# B&R Automation Studio project ABC_Pltzr (part 2)

#### Cyclic.ld
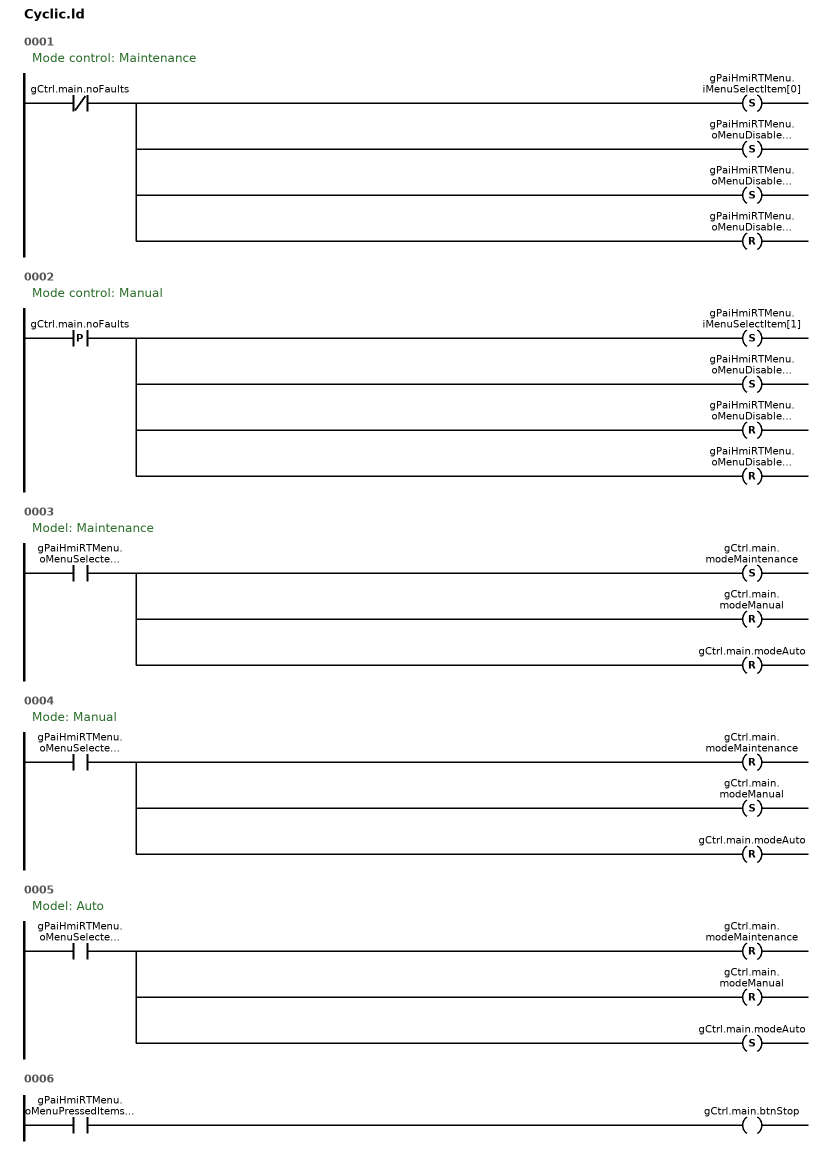
Ladder, written as Structured Text:
```iecst
PROGRAM _CYCLIC
VAR
    _e1 : R_TRIG;
END_VAR
(* Network 1: Mode control: Maintenance *)
IF NOT gCtrl.main.noFaults THEN
    gPaiHmiRTMenu.iMenuSelectItem[0] := TRUE;
    gPaiHmiRTMenu.oMenuDisabledItems[1] := TRUE;
    gPaiHmiRTMenu.oMenuDisabledItems[2] := TRUE;
    gPaiHmiRTMenu.oMenuDisabledItems[0] := FALSE;
END_IF;

(* Network 2: Mode control: Manual *)
_e1(CLK := gCtrl.main.noFaults);
IF _e1.Q THEN
    gPaiHmiRTMenu.iMenuSelectItem[1] := TRUE;
    gPaiHmiRTMenu.oMenuDisabledItems[0] := TRUE;
    gPaiHmiRTMenu.oMenuDisabledItems[1] := FALSE;
    gPaiHmiRTMenu.oMenuDisabledItems[2] := FALSE;
END_IF;

(* Network 3: Model: Maintenance *)
IF gPaiHmiRTMenu.oMenuSelectedItems[0] THEN
    gCtrl.main.modeMaintenance := TRUE;
    gCtrl.main.modeManual := FALSE;
    gCtrl.main.modeAuto := FALSE;
END_IF;

(* Network 4: Mode: Manual *)
IF gPaiHmiRTMenu.oMenuSelectedItems[1] THEN
    gCtrl.main.modeMaintenance := FALSE;
    gCtrl.main.modeManual := TRUE;
    gCtrl.main.modeAuto := FALSE;
END_IF;

(* Network 5: Model: Auto *)
IF gPaiHmiRTMenu.oMenuSelectedItems[2] THEN
    gCtrl.main.modeMaintenance := FALSE;
    gCtrl.main.modeManual := FALSE;
    gCtrl.main.modeAuto := TRUE;
END_IF;

(* Network 6 *)
gCtrl.main.btnStop := gPaiHmiRTMenu.oMenuPressedItems[1];
END_PROGRAM
```

- Program Logical/MachineControl/palletinfauto (IEC) (no source held here)

### Program Logical/paiComponents/bglib

#### bgBitUtilities.h
```c
/**\file: bgBitUtilities.h
*Bit utilities.
*/
#include <bur/plctypes.h>
#ifndef _BG_BITUTILS_H
#define _BG_BITUTILS_H

/**
Set UDINT bits.
\param dest,  Ptr to UDINT.
\param bitIndex within the above UDINT
\param bitValue is the value to set the bit to
*/
void bgBitSetUDINT(UDINT* dest,  UINT bitIndex, BOOL bitValue);

/**
Set UINT bits.
\param dest,  Ptr to UINT.
\param bitIndex within the above UINT
\param bitValue is the value to set the bit to
*/
void bgBitSetUINT(UINT* dest,  UINT bitIndex, BOOL bitValue);

/**
Set USINT bits.
\param dest,  Ptr to USINT.
\param bitIndex within the above USINT
\param bitValue is the value to set the bit to
*/
void bgBitSetUSINT(USINT* dest,  UINT bitIndex, BOOL bitValue);

#endif
```

#### bgPVSerialize.h
```c
/**\file: bgPVSerialize.h
*Serialize/deserialize a PV to/from text stream.
*/
#include <bur/plctypes.h>
#ifndef _BG_PVSERIALIZE_H
#define _BG_PVSERIALIZE_H

/**
Serialize a PV (*pvNameRoot) to an output stream (* toOutStream) with a max length of (lengthOutStream).
\param pvNameRoot ptr to a PV name
\param toOutStream ptr to an output stream (i.e. char buffer)
\param lengthOutStream max length of the output stream in bytes
\return -1 error
\return >=0 number of bytes written to the output stream
*/
DINT bgPVStructSerialize(char* pvNameRoot, char* toOutStream, UDINT lengthOutStream);

/**
Deserialize a PV (*pvNameRoot) from an input stream (* fromStream) that contains (lengthStream) of valid text data.
\param pvNameRoot ptr to a PV name
\param fromStream ptr to an input stream (i.e. char buffer)
\param lengthStream length of the content in the input stream in bytes
\return -1 error
\return >=0 TODO
*/
DINT bgPVStructDeserialize(char* pvNameRoot, char* fromStream, UDINT lengthStream);

/**
Compare two instances of the same structure type using PV services and provide diff report into the given output stream (* toOutStream) with a max length of (lengthOutStream).
\param pvNameRoot ptr to an instance 1 of the PV structure
\param pvNameRoot2 ptr to an instance 2 of the PV structure
\param toOutStream ptr to an output stream (i.e. char buffer)
\param lengthOutStream max length of the output stream in bytes
\return -1 error
\return >=0 number of bytes written to the output stream
*/
DINT bgPVStructCompare(char* pvNameRoot, char* pvNameRoot2, char* toOutStream, UDINT lengthOutStream);

#endif
```

#### bgHttpAppXmlRpc.c
```c
/**\file bgHttpAppXmlRpc.c
*/

#ifndef WIN32
/*
B&R components:
===============================================================================
*/
#include <bur/plc.h>
#include <bur/plctypes.h>
#include <astcp.h>
#include <brsystem.h>
#include <sys_lib.h>
#endif

/*
BG components
===============================================================================
*/
#include "bgdebug.h"
#include "bgstring.h"
#include "bgsscanf.h"
#include "bgTcpSocketClientServer.h"
#include "bgHttpProtocol.h"
#include "bgHttpAppXmlRpc.h"
#include "bgDataStructures.h"
#include "bgBufMemAlloc.h"
#include "bgXmlRpcParser.h"

static void apndXmlBlockOpen(bgTcpSocketSession_typ* pSession, char* keywName);
static void apndXmlBlockClos(bgTcpSocketSession_typ* pSession, char* keywName);

/*
XmlRpc Server
######################################################################################################
######################################################################################################
######################################################################################################
######################################################################################################
*/
void bgXmlRpcServerApplication(bgTcpSocketSession_typ* pSession)
{
char* pMem;
int sizeMem;
char* pMemTree;
int sizeMemTree;
char* pMemStr;
int sizeMemStr;

httpAppXmlRpc_typ* pXmlRpcAppData;
bgXmlRpcParser_typ* pXmlRpc;
bgTree4C_typ* pTree;
bgTree4CNode_typ* pNode;
bgStringHeap_typ* pStrHeap;

int i;

	if( bgXmlRpcServerAppCommon(pSession) ){
		/*common XMLRPC check(s) have failed > exit (& send automatic error response)*/
		return;
	}

/*App Specific Buf MemAlloc*/
	/*1) application specific data structure*/
	if( bgBufMemAllocCreateBlock(&pSession->sessionMem, sizeof(httpAppXmlRpc_typ) + sizeof(char*), &pMem, &sizeMem) )
	{
    	DBGMSG("bgXmlRpcServerApplication(): FATAL ERROR (1); No memory\r\n");
		return;
	}

	pXmlRpcAppData = (httpAppXmlRpc_typ*)pMem;
	pXmlRpc = &pXmlRpcAppData->xmlRpcData;
	pTree = &pXmlRpc->xmlTree;
	pStrHeap = &pXmlRpc->strHeap;

	/*2) set storage for xmlrpc node tree*/
	if( bgBufMemAllocCreateBlock(&pSession->sessionMem, 1500, &pMemTree, &sizeMemTree) )
	{
    	DBGMSG("bgXmlRpcServerApplication(): FATAL ERROR (2); No memory\r\n");
		return;
	}

	/*3) set storage for xmlrpc string heap (rest of the available mem)*/
	if( bgBufMemAllocCreateBlock(&pSession->sessionMem, 0, &pMemStr, &sizeMemStr) )
	{
    	DBGMSG("bgXmlRpcServerApplication(): FATAL ERROR (3); No memory\r\n");
		return;
	}

	DBGMSG("bgXmlRpcServerApplication: memTotal=%d, memData=%d, memTree=%d, memStr=%d\n",
		sizeMem + sizeMemStr + sizeMemTree, sizeMem, sizeMemTree, sizeMemStr);

    bgXmlRpcParserInit(pXmlRpc, bgHttpGetContentStartAddr(pSession), pMemTree, sizeMemTree, pMemStr, sizeMemStr);

    bgXmlRpcParserParse(pXmlRpc);

	if(pXmlRpc->error){
		DBGMSG("xml parsing error=%d; keyword=[%s], line=%d, col=%d)\n",
			pXmlRpc->error,
			bgXmlRpcGetKeywordStr(pXmlRpc->keywId),
			pXmlRpc->keywLineNo,
			pXmlRpc->keywColNo);
/*
			bgXmlRpcServerSendFaultResponse(pSession, 100, "This is fault!");
			rerurn;
*/
	}

    DBGMSG("xmlRpc tree:\n");
    DBGMSG("---------------------------------------------------------------------\n");

    bgTree4CPrint(pTree);

    DBGMSG("---------------------------------------------------------------------\n");

    DBGMSG("xmlRpc list of values:\n");
    DBGMSG("---------------------------------------------------------------------\n");

	for(i=0; i < pTree->nodeCountUsed; i++){

		pNode = &pTree->nodes[i];

		if(!pNode || !pNode->used)
			continue;

		switch(pNode->dataType){
			case XMLRPC_ID_METHOD_NAME:
				DBGMSG("MethodName:[%s]\n", pNode->data ? pNode->data : "unknown");
			break;
			case XMLRPC_ID_NAME:
				DBGMSG("\nParamName:[%s]\n", pNode->data ? pNode->data : "unknown");
			break;
			case XMLRPC_ID_I4:
			case XMLRPC_ID_INT:
			case XMLRPC_ID_BOOL:
				DBGMSG("Value:[%d]\n", pNode->dataValue );

			break;
			case XMLRPC_ID_STRING:
			case XMLRPC_ID_TIME:
				DBGMSG("Value:[%s]\n", pNode->data ? pNode->data : "unknown" );
			break;
			case XMLRPC_ID_DOUBLE:
				DBGMSG("Value:[%f]\n", (float)pNode->dataValue);
			break;
			default:
			break;
		}

	}
    DBGMSG("---------------------------------------------------------------------\n");

	DBGMSG("StringHeap space: total=%d, free=%d\n", pStrHeap->memSize, pStrHeap->memFree );

	bgXmlRpcServerSendFaultResponse(pSession, 100, "This is fault!");
}

int bgXmlRpcServerAppCommon(bgTcpSocketSession_typ* pSession)
{
    /*session/application/protocol specific data structure*/
    httpMessage_typ* r = (httpMessage_typ*)pSession->pProtocol;

	if( r->commandId != BGHTTP_REQUEST_COMMAND_POST){
		DBGMSG("bgXmlRpcServerApplication(): command (%s) not supported!\r\n", r->command);
		bgHttpSendErrorResponse(pSession, 405);
 		return 1;
	}

	return 0;
}

int bgXmlRpcServerSendFaultResponse(bgTcpSocketSession_typ* p, int faultCode, char* faultString)
{
/*
XML-RPC Fault Response Example:

HTTP/1.1 200 OK
Connection: close
Content-Length: 426
Content-Type: text/xml
Date: Fri, 17 Jul 1998 19:55:02 GMT
Server: UserLand Frontier/5.1.2-WinNT

<?xml version="1.0"?>
<methodResponse>
	<fault>
		<value>
			<struct>
				<member>
					<name>faultCode</name>
					<value><int>4</int></value>
				</member>
				<member>
					<name>faultString</name>
					<value><string>Too many parameters.</string></value>
				</member>
			</struct>
		</value>
	</fault>
</methodResponse>
*/
	bgHttpServerSendResponseBeg(p, 200, "text/xml");

	apndXmlBlockOpen(p, XMLRPC_STR_XMLHEADLINE );

	apndXmlBlockOpen(p, XMLRPC_STR_METHOD_RSP);
		apndXmlBlockOpen(p, XMLRPC_STR_FAULT);
			apndXmlBlockOpen(p, XMLRPC_STR_VALUE);
				apndXmlBlockOpen(p, XMLRPC_STR_STRUCT);
					apndXmlBlockOpen(p, XMLRPC_STR_MEMBER);
					{
						char txtBuffer[255];
						bgsprintf(&txtBuffer[0], "<%s>%s</%s>", XMLRPC_STR_NAME, "faultCode", XMLRPC_STR_NAME);
						bgHttpSendBufApndContentLine(p, &txtBuffer[0]);

						bgsprintf(&txtBuffer[0], "<%s><%s>%d</%s></%s>", XMLRPC_STR_VALUE, XMLRPC_STR_INT, faultCode, XMLRPC_STR_INT, XMLRPC_STR_VALUE);
						bgHttpSendBufApndContentLine(p, &txtBuffer[0]);

					}
					apndXmlBlockClos(p, XMLRPC_STR_MEMBER);
					apndXmlBlockOpen(p, XMLRPC_STR_MEMBER);
					{
						char txtBuffer[255];
						bgsprintf(&txtBuffer[0], "<%s>%s</%s>", XMLRPC_STR_NAME, "faultString", XMLRPC_STR_NAME);
						bgHttpSendBufApndContentLine(p, &txtBuffer[0]);

						bgsprintf(&txtBuffer[0], "<%s><%s>%s</%s></%s>", XMLRPC_STR_VALUE, XMLRPC_STR_STRING, faultString, XMLRPC_STR_STRING, XMLRPC_STR_VALUE);
						bgHttpSendBufApndContentLine(p, &txtBuffer[0]);

					}
					apndXmlBlockClos(p, XMLRPC_STR_MEMBER);
				apndXmlBlockClos(p, XMLRPC_STR_STRUCT);
			apndXmlBlockClos(p, XMLRPC_STR_VALUE);
		apndXmlBlockClos(p, XMLRPC_STR_FAULT);
	apndXmlBlockClos(p, XMLRPC_STR_METHOD_RSP );

	bgHttpServerSendResponseEnd(p);
	return 0;
}

int bgXmlRpcServerSendResponse(bgTcpSocketSession_typ* pSession, char* pContent, int contentSize)
{
    bgHttpServerSendResponse(pSession, 200, pContent, contentSize, "text/xml");
	return 0;
}

/*
XmlRpc Client
######################################################################################################
######################################################################################################
######################################################################################################
######################################################################################################
*/
void bgXmlRpcClientSetConnection(bgTcpSocketClient_typ* pClient, char* serverIpAddr, int serverPortNumber)
{
	bgHttpClientSetConnection(pClient, serverIpAddr, serverPortNumber);
}

void bgXmlRpcClientSendRequest(bgTcpSocketClient_typ* pClient, char* pContent , int contentSize)
{
	bgHttpClientSendRequest(pClient, "POST /RPC2 ", pContent , contentSize, "text/xml");
}

void bgXmlRpcClientApplication(bgTcpSocketSession_typ* pSession)
{
int i;
char* pMem;
int sizeMem;
httpAppWeb_typ* pWebData;
int sizeMemAppTotal = 0;

/*App Specific Buf MemAlloc*/
	/*1) application specific data structure*/
	if( bgBufMemAllocCreateBlock(&pSession->sessionMem, sizeof(httpAppWeb_typ) + sizeof(char*), &pMem, &sizeMem) )
	{
    	DBGMSG("bgXmlRpcClientApplication(): FATAL ERROR (1); No memory\r\n");
		return;
	}
	pWebData = (httpAppWeb_typ*)pMem;
	sizeMemAppTotal += sizeMem;

	/*2) set storage for line list (long list of items, i.e. several hundred items, depending on the memory)*/
	if( bgBufMemAllocCreateBlock(&pSession->sessionMem, 0, &pMem, &sizeMem) )
	{
    	DBGMSG("bgXmlRpcClientApplication(): FATAL ERROR (4); No memory\r\n");
		return;
	}
    bgStringListExMemSet(&pWebData->listContentLines, pMem, sizeMem);
	sizeMemAppTotal += sizeMem;
	DBGMSG("bgXmlRpcClientApplication: memTotal=%d, memList=%d\n", sizeMemAppTotal, sizeMem);

	/*if http response does not contain content, request processing is ready*/
	if( !bgHttpGetContentLength(pSession)){
		DBGMSG("bgXmlRpcClientApplication: received response with no content!\n");
		return;
	}

	/*parse content part of the request; generate list of content lines*/
	if( bgStringListLinesEx(&pWebData->listContentLines, bgHttpGetContentStartAddr(pSession), 0, 0) < 0 ){
		DBGMSG("bgXmlRpcClientApplication(): Received content too long! SessionId= %d, len = %d, Error=500\r\n",
			pSession->ident, pSession->rxByteCount);
 		return;
    }

	DBGMSG("bgXmlRpcClientApplication(): Content list (lines=%d):\r\n",
		pWebData->listContentLines.itemCount);
	DBGMSG("============================================\r\n");
	for(i=0;i < pWebData->listContentLines.itemCount;i++){
		DBGMSG("%s\r\n", pWebData->listContentLines.items[i]);
	}
	DBGMSG("============================================\r\n");

 	return;
}
/*
############################################################################################################
*/

static void apndXmlBlockOpen(bgTcpSocketSession_typ* pSession, char* keywName)
{
char txt[255];
	bgsprintf(txt, "<%s>", keywName);
	bgHttpSendBufApndContentLine(pSession, txt);
}

static void apndXmlBlockClos(bgTcpSocketSession_typ* pSession, char* keywName)
{
char txt[255];
	bgsprintf(txt, "</%s>", keywName);
	bgHttpSendBufApndContentLine(pSession, txt);
}
```

- Library Logical/paiComponents/Libraries/sprintf2 (ANSIC) (no source held here)

### paiBnRVFDX64ParRW.typ
```iecst
TYPE
	paiBnRX64ParamItem_typ : 	STRUCT
		oValue : UDINT;
		iValueWR : UDINT;
		iChannelNameRD : STRING[15];
		iChannelNameWR : STRING[15];
		oStatusRD : UDINT;
		oStatusWR : UDINT;
		iMode : UDINT;
		mState : UDINT;
	END_STRUCT;
	paiBnRX64Station_typ : 	STRUCT
		iDeviceName : STRING[31]; (*VFD Device Name (see AsIOAcc library)*)
		iDescription : STRING[31];
		iPtrModuleOk : UDINT; (*ptr to Module OK signal from the drive*)
		mState : UDINT;
		mCurrentEntry : UDINT;
		mMaxValidEntry : UDINT;
		mX64Params : ARRAY[0..paiBnRVFDX64ParamIdxMax]OF paiBnRX64ParamItem_typ; (*list of x64 parameters*)
	END_STRUCT;
	paiBnRVFDX64RWMgr_typ : 	STRUCT
		mState : UDINT;
		mCurrentEntry : UDINT;
		mX64VFDs : ARRAY[0..paiBnRVFDX64DriveIdxMax]OF paiBnRX64Station_typ; (*list of x64 parameters*)
		mAsIOAccRd : AsIOAccRead;
		mAsIOAccWr : AsIOAccWrite;
	END_STRUCT;
END_TYPE
```

- Program Logical/paiComponents/paiFileService/paiFSUnitTest (ANSIC) (no source held here)

### Program Logical/paiComponents/paiHmi

#### paiARSystem.typ
```iecst
(********************************************************************
 * COPYRIGHT --
 ********************************************************************
 * Package: HMI
 * File: cfgPaiArSystem.typ
 * Author: goran
 * Created: October 15, 2014
 ********************************************************************
 * Data types of package HMI
 ********************************************************************)

TYPE
	paiARNetworkAddress_typ : 	STRUCT  (*AR (Automation Runtime) related network settings*)
		ethDevice : STRING[31];
		hostname : STRING[31];
		ipAddr : STRING[15];
		netMask : STRING[15];
		broadcast : STRING[15];
		gateway : STRING[15];
	END_STRUCT;
	paiARSystem_typ : 	STRUCT
		ethernet : paiARNetworkAddress_typ;
	END_STRUCT;
END_TYPE
```

#### paiHmiAlert.typ
```iecst
(********************************************************************
 * COPYRIGHT -- pai
 ********************************************************************
 * Package: HMI
 * File: HMI.typ
 * Author: goran
 * Created: August 28, 2013
 ********************************************************************
 * Data types of package HMI
 ********************************************************************)
(*########################################################################*)
(*HMI object - ALERT*)
(*########################################################################*)

TYPE
	paiHmiAlert_typ : 	STRUCT
		message : STRING[512];
		header : STRING[128];
		type : UINT; (*0-info; 1-warning; 2-error*)
		status : UINT; (*Status for common dialog layer*)
		tmr1RemainingTimeSec : UDINT; (*Timer remaining time (sec)*)
		tmr1 : TON; (*Dialog control timer*)
	END_STRUCT;
END_TYPE
```

#### paiHmiPageChange.h
```c
/********************************************************************
 * COPYRIGHT -- pai
 ********************************************************************
 * Program: hmilogic
 * File: hmiAlert.h
 * Author: goran
 * Created: September 05, 2013
 *******************************************************************/

#include <bur/plctypes.h>
#ifdef _DEFAULT_INCLUDES
#include <AsDefault.h>
#endif
void paiHmiPageChangeInit(paiHmiTemplate_typ* p);
void paiHmiPageChangeCyclic(paiHmiTemplate_typ* p);
```

#### paiHmiDialog.c
```c
/********************************************************************
 * COPYRIGHT -- pai
 ********************************************************************
 * Program: hmilogic
 * File: hmiDialog.c
 * Author: goran
 * Created: September 05, 2013
 *******************************************************************/

#include <bur/plctypes.h>
#ifdef _DEFAULT_INCLUDES
	#include <AsDefault.h>
#endif

/**
Bit manipulaiton utility functions.
 */
#include "../bglib/bgBitUtilities.h"

/**
String manipulaiton utility functions.
 */
//#include <../../bglib/bgsprintf.h>
#include "../bglib/bgstring.h"

/**
 Timer control utility functions.
 */
//#include <../../bglib/bgTimer1ms.h>

/*
###############################################################################
Simple dialog support w. OK and Cancle response
###############################################################################
*/

/**
Find if HMI dialog is active (visible) or not
\param p prt to paiHmiDialog_typ structure
\return 0 not active (not visible)
\return 1 active (visible)
*/
BOOL paiHmiDialogIsActive(paiHmiDialog_typ* p)
{
	//hide the dialog
	if(p->status & 0x1){
		return 0; //not visible > not active
	}

	return 1; //visible > active
}

/**
Hide HMI dialog (make it not visible)
\param p prt to paiHmiDialog_typ structure
*/
void paiHmiDialogHide(paiHmiDialog_typ* p)
{
	//hide the dialog
	bgBitSetUINT(&p->status, 0, 1);

	//define the message
	brsstrcpy((UDINT)p->message, (UDINT)"");
}

/**
Hide HMI dialog (make it not visible)
\param p prt to paiHmiDialog_typ structure
\param msg text message that will be displayed in a dialog
\param timeout_ms time duration to show the dialog. Upon timer expiration, dialog will automatically generate either ok or cancel (configured, see timeoutConfig)
\param resultForOk value returned in case user response is OK (if 0, default is used = 1)
\param resultForCancel value returned in case user response is Cancel ((if 0, default is used = 2)
\param timeoutConfig 0-timeout wil return value for Cancel, 1-timeout will return value for OK
*/
 void paiHmiDialogShow(paiHmiDialog_typ* p, char* msg, UINT timeout_ms, UINT resultForOk, UINT resultForCancel, UINT timeoutConfig)
{
	//show the dialog
	bgBitSetUINT(&p->status, 0, 0);

	//define the message
	bgStrCpyN(p->message, msg, sizeof(p->message));

	//start the timer
	bgTimerStart(&p->tmr1, timeout_ms);

	//set the result to 0 (not complete)
	p->result = 0;

	//configuration of the timeout
	p->timeoutConfig = timeoutConfig;

	p->resultForOk = resultForOk;
	if(!p->resultForOk)
		p->resultForOk = 1;

	p->resultForCancel = resultForCancel;
	if(!p->resultForCancel)
		p->resultForCancel = 2;

}

/**
Hide HMI dialog cyclic routine
\param p prt to paiHmiDialog_typ structure
*/
UINT paiHmiDialogCyclic(paiHmiDialog_typ* p)
{
	//operate timer always
	bgTimerCyclic(&p->tmr1);

	p->tmr1RemainingTimeSec = (p->tmr1.PT - p->tmr1.ET) / 1000;

	//if dialog not visible > nothing to do
	if(p->status)
		return 0;

	if( bgTimerIsTimeOut(&p->tmr1) ){
		//hide the dialog
		paiHmiDialogHide(p);
		//check how is the timeout configured and generate such result
		if(!p->timeoutConfig){
			p->result = p->resultForCancel;
			return p->resultForCancel; //return cancel
		}
		p->result = p->resultForOk;
		return p->resultForOk;//return OK
	}

	//keep checking if the result value will get set by the HMI
	if( p->result ){
		//hide the dialog
		paiHmiDialogHide(p);

		//predefined values in HMI are:
		// 1=OK
		// 2=Cancel
		// Override the above and return what's configured
		if(p->result == 1){
			p->result = p->resultForOk;
		}else{
			p->result = p->resultForCancel;
		}

		return p->result; //return user's choice (1=ok, 2=cancel > see the HMI setup)
	}

	return 0;
}
//EOF
```

- Program Logical/paiComponents/paiMp/paiFileDT (IEC) (no source held here)

### Program Logical/paiComponents/paiTelnet/paiTelnet

#### paiTelnet.c
```c
/********************************************************************
 * COPYRIGHT --
 ********************************************************************
 * Program: paiTelnet
 * File: paiTelnet.c
 * Author: goran
 * Created: June 23, 2015
 ********************************************************************
 * Implementation of program paiTelnet
 ********************************************************************/

#include <bur/plctypes.h>

#ifdef _DEFAULT_INCLUDES
	#include <AsDefault.h>
#endif

//#include "../../bglib/bgringbuffer.h"
#include "../../libraries/bgringbuf/bgringbuffer.h"
#include "../../bglib/bgTelnetSrvr-astcpV2.h"

_GLOBAL bgRingBuffer_typ gRingBuffer;

void _INIT paiTelnetInit(void)
{
//	DefineRingBuff(&gRingBuffer);

	/* TODO: Add code here */
	bgTelnetSrvrInit(&dbgTerm, &gRingBuffer);

}

void _CYCLIC paiTelnetCyclic(void)
{
	/* TODO: Add code here */
	bgTelnetSrvrCyclic(&dbgTerm);
}
```

### paiConfigSys.typ
```iecst
(********************************************************************
 * COPYRIGHT --
 ********************************************************************
 * Package: paiHMI
 * File: paiConfigSys.typ
 * Author: goran_2
 * Created: August 06, 2011
 ********************************************************************
 * Data types of package paiComponents
 ********************************************************************)

TYPE
	paiConfigSystem_typ : 	STRUCT  (*Generic (System) configuration defined by PAI*)
		paiSys : paiARSystem_typ;
	END_STRUCT;
END_TYPE
```

### paiHMI.typ
```iecst
(********************************************************************
 * COPYRIGHT -- pai
 ********************************************************************
 * Package: HMI
 * File: HMI.typ
 * Author: goran
 * Created: August 28, 2013
 ********************************************************************
 * Data types of package HMI
 ********************************************************************)

TYPE
	hmiControlLogicEnums_typ :
		(
		hmiREMMEM_MAGIC := 16#55555555, (*Magic number*)
		hmiSecurityHMIUsersMAXIDX := 11, (*Max number of HMI users - 1*)
		hmiLoggerPVCmpBufSize := 2047, (*Size of the PV compare buffer*)
		HMI_ENUM_TAB_KEYS_MAX := 10, (*Max number of tab keys per page*)
		HMI_PWD_LEVELS := 5, (*Number of password levels (0-operator;1-supervisor;2-admin;3-maintenance;4-factory)*)
		HMI_PWD_MAXLEN := 15 (*Max pwd len*)
		);
END_TYPE

(*########################################################################*)
(*Application object - Security Manager*)
(*########################################################################*)

TYPE
	hmiSecurityUser_typ : 	STRUCT
		loginLevel : UDINT; (*0-operator (no HMI access);1-supervisor;2-admin;3-maintenance;4-GAINCO*)
		userPIN : STRING[7];
		userName : STRING[63];
	END_STRUCT;
	hmiSecurityManager_typ : 	STRUCT
		webSecurityActive : UDINT;
		dbUpdateEvent : UDINT;
		visibleIfUserSecurityActive : UDINT;
		visibleIfUserSecurityNOTActive : UDINT;
		userIsLoggedIn : UDINT;
		loggedInUserIdx : UDINT;
		hmiUserIndex : UDINT;
		hmiUserIndexMax : UDINT;
		hmiPINSelected : UDINT;
		hmiPINCompletion : UDINT;
		hmiLoggedUserName : STRING[63];
		hmiListOfUserPINs : ARRAY[0..hmiSecurityHMIUsersMAXIDX]OF STRING[7];
		hmiListOfUserNames : ARRAY[0..hmiSecurityHMIUsersMAXIDX]OF STRING[63];
		listOfUsers : ARRAY[0..hmiSecurityHMIUsersMAXIDX]OF hmiSecurityUser_typ;
	END_STRUCT;
END_TYPE

(*########################################################################*)
(*Application object - Event Logger Manager*)
(*########################################################################*)

TYPE
	hmiEventLoggerManager_typ : 	STRUCT
		pvCompareEvent : UDINT; (*Set to 1 when MachineCfg strucutres changes. Allows logger manager to capture changed values and send them to DB.*)
		pvCompareResult : INT;
		pvCompareBuf : STRING[hmiLoggerPVCmpBufSize];
	END_STRUCT;
END_TYPE
```

- Visualisation Logical/paiComponents/paiTemplate/paiHMI/paiScreens/paXGA (not shown)

- Program Logical/paiComponents/paiUDP/udpApp (ANSIC) - pai UDP Service (TK#8) (no source held here)

### Package Logical/ParameterDownload/X64_S44_Download - download the parameters from the X64

### Program Logical/ParameterDownload/X64_S44_Download/S44param (IEC)

#### S44paramInit.st - Initialization code
```iecst
(********************************************************************
 * COPYRIGHT --
 ********************************************************************
 * Program: S44param
 * File: S44paramInit.st
 * Author: scoccimaroj
 * Created: July 15, 2010
 ********************************************************************
 * Implementation of program S44param
 ********************************************************************)

PROGRAM _INIT

strcpy( ADR(S44ParRead.pDevice) , ADR('SS1.IF1.ST1') );
AsIOAccRead_0.pDeviceName := ADR(S44ParRead.pDevice);
strcpy( ADR(S44ParRead.FileDevice), ADR('DISK') );

 (* Initialize the CSV file writing operation *)
 strcpy( ADR(S44ParRead.CsvFileName), ADR(S44ParRead.pDevice) );

 FOR i:= 0 TO 10 BY 1 DO
 	position := FIND(S44ParRead.CsvFileName, '.');

	IF (position <> 0) THEN
 		S44ParRead.CsvFileName := REPLACE(S44ParRead.CsvFileName, '_', 1, position);
	END_IF

 END_FOR

 strcat( ADR(S44ParRead.CsvFileName), ADR('.csv') );

 pNames[0] := ADR('S44ParRead');

 csvInit.pStructName := ADR(pNames);
 csvInit.NumOfStructs := 1;
 csvInit.FullNameLenght := 0;
 csvInit.Options := 0;

 csvInit();

 IF (csvInit.status = 0) THEN
 	csvMemLength := csvInit.MemCounter;
	csvStrucMem := csvInit.pStructMem;

	csvInitCheckFile.MemCounter := csvMemLength;
	csvInitCheckFile.enable := 1;
	csvInitCheckFile();

 END_IF

(* Initialize the parameter channel names *)
strcpy( ADR(S44ParRead.Parameters[0].ChannelName) , ADR('COD_Input') );
strcpy( ADR(S44ParRead.Parameters[1].ChannelName) , ADR('BFR_Input') );
strcpy( ADR(S44ParRead.Parameters[2].ChannelName) , ADR('FR1_Input') );
strcpy( ADR(S44ParRead.Parameters[3].ChannelName) , ADR('ACC_Input') );
strcpy( ADR(S44ParRead.Parameters[4].ChannelName) , ADR('DEC_Input') );
strcpy( ADR(S44ParRead.Parameters[5].ChannelName) , ADR('LSP_Input') );
strcpy( ADR(S44ParRead.Parameters[6].ChannelName) , ADR('HSP_Input') );
strcpy( ADR(S44ParRead.Parameters[7].ChannelName) , ADR('NPR_Input') );
strcpy( ADR(S44ParRead.Parameters[8].ChannelName) , ADR('NCR_Input') );
strcpy( ADR(S44ParRead.Parameters[9].ChannelName) , ADR('AI1T_Input') );
strcpy( ADR(S44ParRead.Parameters[10].ChannelName) , ADR('TCC_Input') );
strcpy( ADR(S44ParRead.Parameters[11].ChannelName) , ADR('TCT_Input') );
strcpy( ADR(S44ParRead.Parameters[12].ChannelName) , ADR('NPL_Input') );
strcpy( ADR(S44ParRead.Parameters[13].ChannelName) , ADR('CRL1_Input') );
strcpy( ADR(S44ParRead.Parameters[14].ChannelName) , ADR('CRH1_Input') );
strcpy( ADR(S44ParRead.Parameters[15].ChannelName) , ADR('R1_Input') );
strcpy( ADR(S44ParRead.Parameters[16].ChannelName) , ADR('LO1_Input') );
strcpy( ADR(S44ParRead.Parameters[17].ChannelName) , ADR('LO1S_Input') );
strcpy( ADR(S44ParRead.Parameters[18].ChannelName) , ADR('TOL_Input') );
strcpy( ADR(S44ParRead.Parameters[19].ChannelName) , ADR('LOC_Input') );
strcpy( ADR(S44ParRead.Parameters[20].ChannelName) , ADR('ULT_Input') );
strcpy( ADR(S44ParRead.Parameters[21].ChannelName) , ADR('LUL_Input') );
strcpy( ADR(S44ParRead.Parameters[22].ChannelName) , ADR('FTD_Input') );
strcpy( ADR(S44ParRead.Parameters[23].ChannelName) , ADR('CTD_Input') );
strcpy( ADR(S44ParRead.Parameters[24].ChannelName) , ADR('TTD_Input') );
strcpy( ADR(S44ParRead.Parameters[25].ChannelName) , ADR('AO1_Input') );
strcpy( ADR(S44ParRead.Parameters[26].ChannelName) , ADR('AO1T_Input') );
strcpy( ADR(S44ParRead.Parameters[27].ChannelName) , ADR('COS_Input') );
strcpy( ADR(S44ParRead.Parameters[28].ChannelName) , ADR('UNS_Input') );
strcpy( ADR(S44ParRead.Parameters[29].ChannelName) , ADR('FRS_Input') );
strcpy( ADR(S44ParRead.Parameters[30].ChannelName) , ADR('NSP_Input') );
strcpy( ADR(S44ParRead.Parameters[31].ChannelName) , ADR('TFR_Input') );
strcpy( ADR(S44ParRead.Parameters[32].ChannelName) , ADR('CTT_Input') );
strcpy( ADR(S44ParRead.Parameters[33].ChannelName) , ADR('UFR_Input') );
strcpy( ADR(S44ParRead.Parameters[34].ChannelName) , ADR('SLP_Input') );
strcpy( ADR(S44ParRead.Parameters[35].ChannelName) , ADR('STA_Input') );
strcpy( ADR(S44ParRead.Parameters[36].ChannelName) , ADR('FLG_Input') );
strcpy( ADR(S44ParRead.Parameters[37].ChannelName) , ADR('PFL_Input') );
strcpy( ADR(S44ParRead.Parameters[38].ChannelName) , ADR('SFR_Input') );
strcpy( ADR(S44ParRead.Parameters[39].ChannelName) , ADR('SFT_Input') );
strcpy( ADR(S44ParRead.Parameters[40].ChannelName) , ADR('NRD_Input') );
strcpy( ADR(S44ParRead.Parameters[41].ChannelName) , ADR('TUN_Input') );
strcpy( ADR(S44ParRead.Parameters[42].ChannelName) , ADR('MPC_Input') );
strcpy( ADR(S44ParRead.Parameters[43].ChannelName) , ADR('RIN_Input') );
strcpy( ADR(S44ParRead.Parameters[44].ChannelName) , ADR('PST_Input') );
strcpy( ADR(S44ParRead.Parameters[45].ChannelName) , ADR('CHCF_Input') );
strcpy( ADR(S44ParRead.Parameters[46].ChannelName) , ADR('CD1_Input') );
strcpy( ADR(S44ParRead.Parameters[47].ChannelName) , ADR('FLO_Input') );
strcpy( ADR(S44ParRead.Parameters[48].ChannelName) , ADR('FLOC_Input') );
strcpy( ADR(S44ParRead.Parameters[49].ChannelName) , ADR('RPT_Input') );
strcpy( ADR(S44ParRead.Parameters[50].ChannelName) , ADR('RPS_Input') );
strcpy( ADR(S44ParRead.Parameters[51].ChannelName) , ADR('AC2_Input') );
strcpy( ADR(S44ParRead.Parameters[52].ChannelName) , ADR('DE2_Input') );
strcpy( ADR(S44ParRead.Parameters[53].ChannelName) , ADR('BRA_Input') );
strcpy( ADR(S44ParRead.Parameters[54].ChannelName) , ADR('STT_Input') );
strcpy( ADR(S44ParRead.Parameters[55].ChannelName) , ADR('NST_Input') );
strcpy( ADR(S44ParRead.Parameters[56].ChannelName) , ADR('FST_Input') );
strcpy( ADR(S44ParRead.Parameters[57].ChannelName) , ADR('DCF_Input') );
strcpy( ADR(S44ParRead.Parameters[58].ChannelName) , ADR('RRS_Input') );
strcpy( ADR(S44ParRead.Parameters[59].ChannelName) , ADR('ADC_Input') );
strcpy( ADR(S44ParRead.Parameters[60].ChannelName) , ADR('SDC1_Input') );
strcpy( ADR(S44ParRead.Parameters[61].ChannelName) , ADR('TDC1_Input') );
strcpy( ADR(S44ParRead.Parameters[62].ChannelName) , ADR('JOG_Input') );
strcpy( ADR(S44ParRead.Parameters[63].ChannelName) , ADR('PS2_Input') );
strcpy( ADR(S44ParRead.Parameters[64].ChannelName) , ADR('PS4_Input') );
strcpy( ADR(S44ParRead.Parameters[65].ChannelName) , ADR('PS8_Input') );
strcpy( ADR(S44ParRead.Parameters[66].ChannelName) , ADR('SP2_Input') );
strcpy( ADR(S44ParRead.Parameters[67].ChannelName) , ADR('SP3_Input') );
strcpy( ADR(S44ParRead.Parameters[68].ChannelName) , ADR('SP4_Input') );
strcpy( ADR(S44ParRead.Parameters[69].ChannelName) , ADR('SP5_Input') );
strcpy( ADR(S44ParRead.Parameters[70].ChannelName) , ADR('SP6_Input') );
strcpy( ADR(S44ParRead.Parameters[71].ChannelName) , ADR('SP7_Input') );
strcpy( ADR(S44ParRead.Parameters[72].ChannelName) , ADR('SP8_Input') );
strcpy( ADR(S44ParRead.Parameters[73].ChannelName) , ADR('JPF_Input') );
strcpy( ADR(S44ParRead.Parameters[74].ChannelName) , ADR('PIF_Input') );
strcpy( ADR(S44ParRead.Parameters[75].ChannelName) , ADR('RPG_Input') );
strcpy( ADR(S44ParRead.Parameters[76].ChannelName) , ADR('RIG_Input') );
strcpy( ADR(S44ParRead.Parameters[77].ChannelName) , ADR('RDG_Input') );
strcpy( ADR(S44ParRead.Parameters[78].ChannelName) , ADR('FBS_Input') );
strcpy( ADR(S44ParRead.Parameters[79].ChannelName) , ADR('PII_Input') );
strcpy( ADR(S44ParRead.Parameters[80].ChannelName) , ADR('PR2_Input') );
strcpy( ADR(S44ParRead.Parameters[81].ChannelName) , ADR('PR4_Input') );
strcpy( ADR(S44ParRead.Parameters[82].ChannelName) , ADR('RP2_Input') );
strcpy( ADR(S44ParRead.Parameters[83].ChannelName) , ADR('RP3_Input') );
strcpy( ADR(S44ParRead.Parameters[84].ChannelName) , ADR('RP4_Input') );
strcpy( ADR(S44ParRead.Parameters[85].ChannelName) , ADR('RPI_Input') );
strcpy( ADR(S44ParRead.Parameters[86].ChannelName) , ADR('PRP_Input') );
strcpy( ADR(S44ParRead.Parameters[87].ChannelName) , ADR('RPL_Input') );
strcpy( ADR(S44ParRead.Parameters[88].ChannelName) , ADR('RPH_Input') );
strcpy( ADR(S44ParRead.Parameters[89].ChannelName) , ADR('SFS_Input') );
strcpy( ADR(S44ParRead.Parameters[90].ChannelName) , ADR('PIC_Input') );
strcpy( ADR(S44ParRead.Parameters[91].ChannelName) , ADR('PAU_Input') );
strcpy( ADR(S44ParRead.Parameters[92].ChannelName) , ADR('PIM_Input') );
strcpy( ADR(S44ParRead.Parameters[93].ChannelName) , ADR('RSL_Input') );
strcpy( ADR(S44ParRead.Parameters[94].ChannelName) , ADR('UPP_Input') );
strcpy( ADR(S44ParRead.Parameters[95].ChannelName) , ADR('LC2_Input') );
strcpy( ADR(S44ParRead.Parameters[96].ChannelName) , ADR('CLI_Input') );
strcpy( ADR(S44ParRead.Parameters[97].ChannelName) , ADR('CL2_Input') );
strcpy( ADR(S44ParRead.Parameters[98].ChannelName) , ADR('TLS_Input') );
strcpy( ADR(S44ParRead.Parameters[99].ChannelName) , ADR('SH2_Input') );
strcpy( ADR(S44ParRead.Parameters[100].ChannelName) , ADR('SH4_Input') );
strcpy( ADR(S44ParRead.Parameters[101].ChannelName) , ADR('HSP2_Input') );
strcpy( ADR(S44ParRead.Parameters[102].ChannelName) , ADR('HSP3_Input') );
strcpy( ADR(S44ParRead.Parameters[103].ChannelName) , ADR('HSP4_Input') );
strcpy( ADR(S44ParRead.Parameters[104].ChannelName) , ADR('RSF_Input') );
strcpy( ADR(S44ParRead.Parameters[105].ChannelName) , ADR('ATR_Input') );
strcpy( ADR(S44ParRead.Parameters[106].ChannelName) , ADR('TAR_Input') );
strcpy( ADR(S44ParRead.Parameters[107].ChannelName) , ADR('FLR_Input') );
strcpy( ADR(S44ParRead.Parameters[108].ChannelName) , ADR('ITH_Input') );
strcpy( ADR(S44ParRead.Parameters[109].ChannelName) , ADR('THT_Input') );
strcpy( ADR(S44ParRead.Parameters[110].ChannelName) , ADR('OLL_Input') );
strcpy( ADR(S44ParRead.Parameters[111].ChannelName) , ADR('MTM_Input') );
strcpy( ADR(S44ParRead.Parameters[112].ChannelName) , ADR('OPL_Input') );
strcpy( ADR(S44ParRead.Parameters[113].ChannelName) , ADR('IPL_Input') );
strcpy( ADR(S44ParRead.Parameters[114].ChannelName) , ADR('USB_Input') );
strcpy( ADR(S44ParRead.Parameters[115].ChannelName) , ADR('STP_Input') );
strcpy( ADR(S44ParRead.Parameters[116].ChannelName) , ADR('STM_Input') );
strcpy( ADR(S44ParRead.Parameters[117].ChannelName) , ADR('STRT_Input') );
strcpy( ADR(S44ParRead.Parameters[118].ChannelName) , ADR('LFL_Input') );
strcpy( ADR(S44ParRead.Parameters[119].ChannelName) , ADR('INH_Input') );
strcpy( ADR(S44ParRead.Parameters[120].ChannelName) , ADR('SLL_Input') );
strcpy( ADR(S44ParRead.Parameters[121].ChannelName) , ADR('DRN_Input') );
strcpy( ADR(S44ParRead.Parameters[122].ChannelName) , ADR('TTO_Input') );

END_PROGRAM
```

### Program Logical/ParameterDownload/X64_S44_Download/X64param

#### X64paramCyclic.st
```iecst
(********************************************************************
 * COPYRIGHT --
 ********************************************************************
 * Program: X64param
 * File: X64paramCyclic.st
 * Author: scoccimaroj
 * Created: July 14, 2010
 ********************************************************************
 * Implementation of program X64param
 ********************************************************************)

PROGRAM _CYCLIC

CASE State OF

	(* Wait for a start command *)
	0:

		IF (cmdStart) THEN
			cmdStart :=	0;
			i := 0;
			State := 1;
		END_IF

	(* Reads the X64 parameter *)
	1:
		AsIOAccRead_0.enable :=	1;
		AsIOAccRead_0.pChannelName := ADR(X64ParRead.Parameters[i].ChannelName);

		(* If the status = 0, then the read was successful.  Store the value read. *)
		IF (AsIOAccRead_0.status = 0) THEN
			X64ParRead.Parameters[i].Data := AsIOAccRead_0.value;
			AsIOAccRead_0.enable :=	0;
			State := 2;

		(* Remain until the Read FUB is completed *)
		ELSIF (AsIOAccRead_0.status = ERR_FUB_BUSY) OR (AsIOAccRead_0.status = ERR_FUB_ENABLE_FALSE) THEN
			State := 1;

		(* If a FUB error occurs go to the next parameter *)
		ELSE
			AsIOAccRead_0.enable :=	0;
			State := 2;
		END_IF

	2:
		(* all the parameters have been read *)
		IF (i >= NUM_OF_X64PAR) THEN
  			i := 0;
			State := 3;

		(* read the next parameter in the list *)
		ELSE
			i := i + 1;
			State := 1;

		END_IF

	(* Do a csv search to allocate memory for the csv file. *)
	3:
		csvSearch.pStructName := csvInit.pStructName;
		csvSearch.NumOfStructs := csvInit.NumOfStructs;
		csvSearch.pStructMem := csvInit.pStructMem;
		csvSearch.MemLen := csvInit.MemCounter;
		csvSearch.FullNameLenght := 0;
		csvSearch.Separator := 44; (* ascii code for , *)
		csvSearch.Options := 0;
		csvSearch.FileHeader := HEADER;
		csvSearch.pMaschineNo := ADR('machine 1');
  		csvSearch.pComment := ADR('X64 parameter read file');
  		csvSearch.pVersion := ADR('v0.01');
  		csvSearch();

		(* successfully created the file for writing *)
		IF (csvSearch.status = 0) THEN
			State := 4;

		(* Error occured to abort the process *)
		ELSIF (csvSearch.status <> 0) AND (csvSearch.status <> 65535) THEN
			State := 0;

		END_IF

	(* Write the data to the csv file *)
	4:
		csvWrite.pFileName := ADR(X64ParRead.CsvFileName);
  		csvWrite.pDevice := ADR(X64ParRead.FileDevice);
  		csvWrite.pPath := ADR(X64ParRead.FilePath);
  		csvWrite.pStructMem := csvInit.pStructMem;
		csvWrite.MemLen := csvSearch.FileLen;
		csvWrite.Mode := FILE_OW;
		csvWrite();

		(* Write completed successfully *)
		IF (csvWrite.status = 0) THEN
  			State := 0;

		ELSIF (csvWrite.status <> 0) AND (csvWrite.status <> 65535) THEN
			State := 0;

		END_IF

END_CASE

(* Function Block Calls *)
AsIOAccRead_0();

END_PROGRAM
```

### Library Logical/ParameterDownload/CSV_File (IEC)
